# EPICS substitutions: iocBoot/ioczzz/asynRecord.substitutions
file "$(ASYN)/db/asynRecord.db"
{
pattern
{P        R         PORT    ADDR    OMAX  IMAX}
{zzz:     asyn_1   serial1    0     256  256}
{zzz:     asyn_2   serial2    0     256  256}
{zzz:     asyn_3   serial3    0     256  256}
{zzz:     asyn_4   serial4    0     256  256}
}
